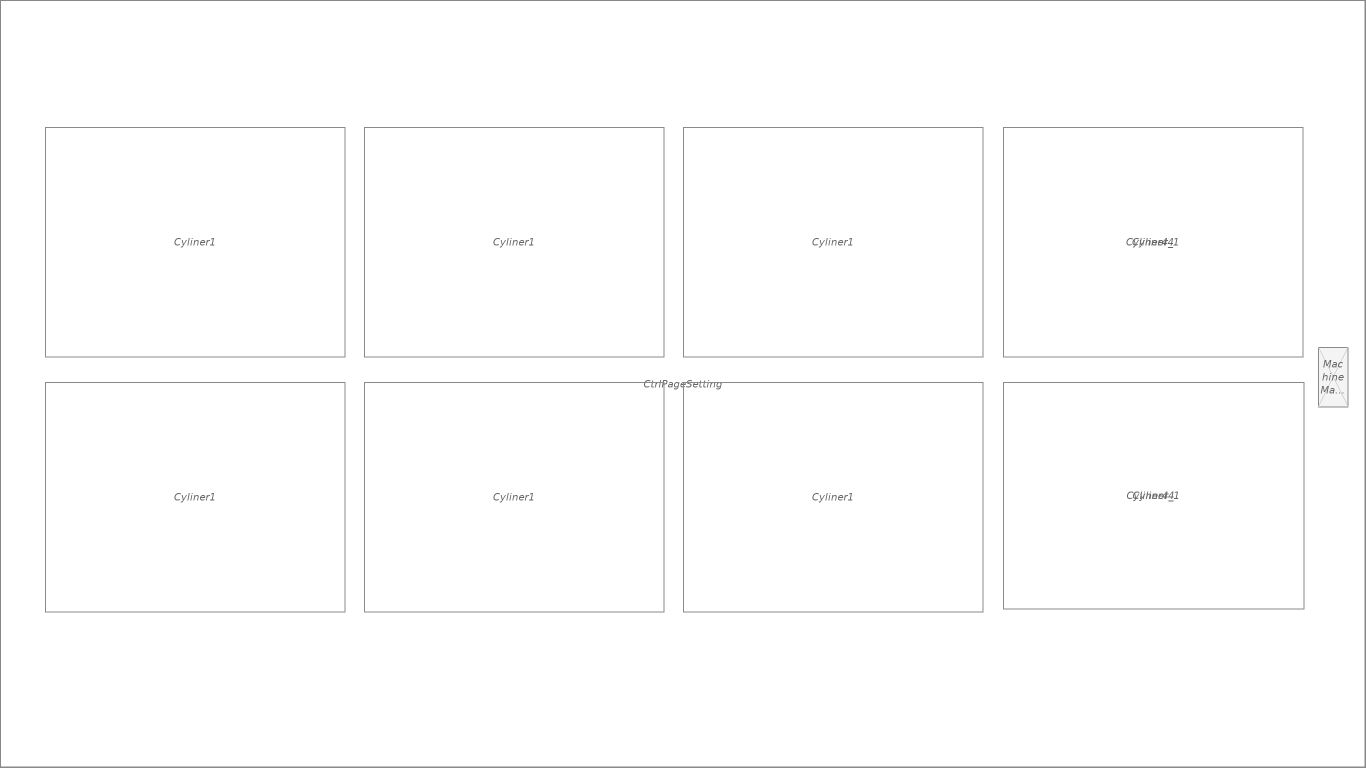
VISUALIZATION PageSetting_OpenLock  // 1366x768
    Frame (0,0 1366x768)
        shows CtrlPageSetting()
    Frame (1003,127 300x230), invisible if: GVL_Data.stRecipe.eProductType<>E_ProductType.Right or GVL_Data.stRecipe.eMachineType<> E_MachineType._311
        shows Cyliner4_1(System := G_stSystem, Cylinder := G_arrCylinder[E_Cylinder.OpenLockRotate], CylinderData := G_arrCylinderData[E_Cylinder.OpenLockRotate])
    Frame (45,127 300x230)
        shows Cyliner1(System := G_stSystem, Cylinder := G_arrCylinder[E_Cylinder.OpenLockPrevent], CylinderData := G_arrCylinderData[E_Cylinder.OpenLockPrevent])
    Frame (364,127 300x230)
        shows Cyliner1(System := G_stSystem, Cylinder := G_arrCylinder[E_Cylinder.OpenLockLift], CylinderData := G_arrCylinderData[E_Cylinder.OpenLockLift])
    Frame (683,127 300x230)
        shows Cyliner1(System := G_stSystem, Cylinder := G_arrCylinder[E_Cylinder.OpenLockPush], CylinderData := G_arrCylinderData[E_Cylinder.OpenLockPush])
    Frame (1003,127 300x230), invisible if: GVL_Data.stRecipe.eProductType<>E_ProductType.Left and GVL_Data.stRecipe.eMachineType= E_MachineType._311
        shows Cyliner4(System := G_stSystem, Cylinder := G_arrCylinder[E_Cylinder.OpenLockRotate], CylinderData := G_arrCylinderData[E_Cylinder.OpenLockRotate])
    Frame (45,382 300x230)
        shows Cyliner1(System := G_stSystem, Cylinder := G_arrCylinder[E_Cylinder.OpenLockPush2], CylinderData := G_arrCylinderData[E_Cylinder.OpenLockPush2])
    Frame (1003,382 301x227), invisible if: GVL_Data.stRecipe.eProductType<>E_ProductType.Right or GVL_Data.stRecipe.eMachineType<> E_MachineType._311
        shows Cyliner4_1(System := G_stSystem, Cylinder := G_arrCylinder[E_Cylinder.OpenLockTranslation], CylinderData := G_arrCylinderData[E_Cylinder.OpenLockTranslation])
    Frame (1003,382 301x227)
        shows Cyliner4(System := G_stSystem, Cylinder := G_arrCylinder[E_Cylinder.OpenLockTranslation], CylinderData := G_arrCylinderData[E_Cylinder.OpenLockTranslation])
    Frame (364,382 300x230)
        shows Cyliner1(System := G_stSystem, Cylinder := G_arrCylinder[E_Cylinder.OpenLockElevator], CylinderData := G_arrCylinderData[E_Cylinder.OpenLockElevator])
    Frame (683,382 300x230)
        shows Cyliner1(System := G_stSystem, Cylinder := G_arrCylinder[E_Cylinder.OpenLockPin], CylinderData := G_arrCylinderData[E_Cylinder.OpenLockPin])
    Image (1318,347 30x60), image: MachineManage.ImagePool.next
        OnMouseClick: change screen: PageSetting_OpenLock_2
END_VISUALIZATION

(* stored: Version 1.1.0.1, ProductVersion 3.1.4024.3
   Visu PageSetting_OpenLock: Id {a58f5456-975f-48d1-b48c-097c5fb8825d} *)
